Staubli VAL3: initParams.pgx

public program initParams()
begin
  nRetVal=sioCtrl(siTcpIpFbk,"port",11002)
  if (nRetVal!=0)
    popUpMsg("Error while setting IP port")
    //return ?
  endIf

  nRetVal=sioCtrl(siTcpIpFbk,"timeout",5)
  if (nRetVal!=0)
    popUpMsg("Error while setting TCP/IP timeout")
    //return ?
  endIf
end
